{attribute 'qualified_only'}
// Robot6 Data
VAR_GLOBAL CONSTANT
	(* cart joints are defiend in sequence as below
	[monitor lift, monitor rotate, armset, pedal] *)
	
	// absolute encoder value at minimal joint positon
	g_minLinkEncoder :ARRAY[1..4] OF DINT :=[8324215, 3073088, 9822199,5580000];
		 
	// absolute encoder value at maximum joint positon
	g_maxLinkEncoder :ARRAY[1..4] OF DINT :=[6650464, 15542320,8563889,6455968];
	
	// absolute encoder value at calibrated positon
	g_caliLinkEncoder :ARRAY[1..4] OF DINT :=[8324215, 3073088, 9822199, 5580000];
	
	// if absolute encoder value cross zeros within joint motion range
	g_linkEncZeroCross :ARRAY[1..4] OF INT :=[0, 0, 0, 0];
	
	 //################ DO NOT modify parameters below ###########################
	// abolute encoder expanded limit buffer in case there is calibrtion error at limit position
	g_linkEncLimitBuffer : DINT := 100000;
	
	// flag if joint can rotate multiple cycles
	g_multipleCyclesJoint :ARRAY[1..4] OF INT :=[0, 0, 0, 0];
		 
	// joint position at link encoder calibrated point
	//TODO: joint2 calibration position need to be checked
	g_linkEncCaliJntPos :ARRAY[1..4] OF LREAL :=[0, 0,0,0];

END_VAR

(* stored: Version 1.1.0.1, ProductVersion 3.1.4024.12
   GVL GVL_CartJointCaliData_6: Id {bd3edc3f-c214-41bd-884d-bc19b98011e2} *)
